% RSLogix 500 project I2P Hands-On 4 - Myah.RSS, saved by version 10.00.00.00 %
PROJECT "UNTITLED"    % processor: Bul.1763 MicroLogix 1100 Series B %

PROGRAM FILES
  LAD 2   15 rungs

DATA FILES
  O0 OUTPUT  4 elements
  I1 INPUT  6 elements
  S2 STATUS  66 elements
  B3 BINARY  1 elements
  T4 TIMER  1 elements
  C5 COUNTER  1 elements
  R6 CONTROL  1 elements
  N7 INTEGER  1 elements
  F8 FLOAT  1 elements

LADDER 2
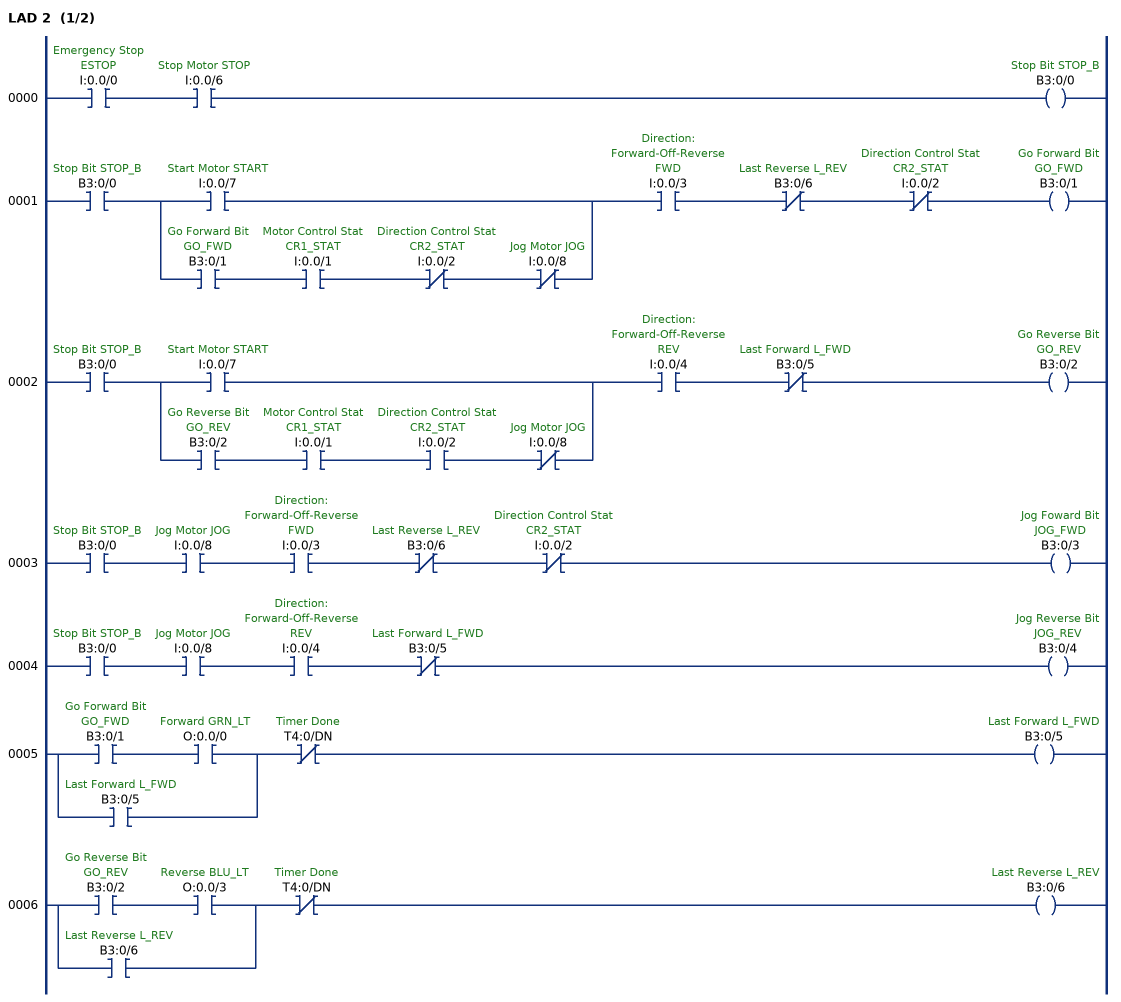
% Rung: 0 %
SOR XIC I:0.0/0 XIC I:0.0/6 OTE B3:0/0 EOR
%   I:0.0/0  ESTOP  "Emergency Stop" %
%   I:0.0/6  STOP  "Stop Motor" %
%   B3:0/0  STOP_B  "Stop Bit" %
% Rung: 1 %
SOR XIC B3:0/0 BST XIC I:0.0/7 NXB XIC B3:0/1 XIC I:0.0/1 XIO I:0.0/2 XIO I:0.0/8 BND XIC I:0.0/3 XIO B3:0/6 XIO I:0.0/2 OTE B3:0/1 EOR
%   B3:0/0  STOP_B  "Stop Bit" %
%   I:0.0/7  START  "Start Motor" %
%   B3:0/1  GO_FWD  "Go Forward Bit" %
%   I:0.0/1  CR1_STAT  "Motor Control Stat" %
%   I:0.0/2  CR2_STAT  "Direction Control Stat" %
%   I:0.0/8  JOG  "Jog Motor" %
%   I:0.0/3  FWD  "Direction: Forward-Off-Reverse" %
%   B3:0/6  L_REV  "Last Reverse" %
% Rung: 2 %
SOR XIC B3:0/0 BST XIC I:0.0/7 NXB XIC B3:0/2 XIC I:0.0/1 XIC I:0.0/2 XIO I:0.0/8 BND XIC I:0.0/4 XIO B3:0/5 OTE B3:0/2 EOR
%   B3:0/0  STOP_B  "Stop Bit" %
%   I:0.0/7  START  "Start Motor" %
%   B3:0/2  GO_REV  "Go Reverse Bit" %
%   I:0.0/1  CR1_STAT  "Motor Control Stat" %
%   I:0.0/2  CR2_STAT  "Direction Control Stat" %
%   I:0.0/8  JOG  "Jog Motor" %
%   I:0.0/4  REV  "Direction: Forward-Off-Reverse" %
%   B3:0/5  L_FWD  "Last Forward" %
% Rung: 3 %
SOR XIC B3:0/0 XIC I:0.0/8 XIC I:0.0/3 XIO B3:0/6 XIO I:0.0/2 OTE B3:0/3 EOR
%   B3:0/0  STOP_B  "Stop Bit" %
%   I:0.0/8  JOG  "Jog Motor" %
%   I:0.0/3  FWD  "Direction: Forward-Off-Reverse" %
%   B3:0/6  L_REV  "Last Reverse" %
%   I:0.0/2  CR2_STAT  "Direction Control Stat" %
%   B3:0/3  JOG_FWD  "Jog Foward Bit" %
% Rung: 4 %
SOR XIC B3:0/0 XIC I:0.0/8 XIC I:0.0/4 XIO B3:0/5 OTE B3:0/4 EOR
%   B3:0/0  STOP_B  "Stop Bit" %
%   I:0.0/8  JOG  "Jog Motor" %
%   I:0.0/4  REV  "Direction: Forward-Off-Reverse" %
%   B3:0/5  L_FWD  "Last Forward" %
%   B3:0/4  JOG_REV  "Jog Reverse Bit" %
% Rung: 5 %
SOR BST XIC B3:0/1 XIC O:0.0/0 NXB XIC B3:0/5 BND XIO T4:0/DN OTE B3:0/5 EOR
%   B3:0/1  GO_FWD  "Go Forward Bit" %
%   O:0.0/0  GRN_LT  "Forward" %
%   B3:0/5  L_FWD  "Last Forward" %
%   T4:0/DN  "Timer Done" %
% Rung: 6 %
SOR BST XIC B3:0/2 XIC O:0.0/3 NXB XIC B3:0/6 BND XIO T4:0/DN OTE B3:0/6 EOR
%   B3:0/2  GO_REV  "Go Reverse Bit" %
%   O:0.0/3  BLU_LT  "Reverse" %
%   B3:0/6  L_REV  "Last Reverse" %
%   T4:0/DN  "Timer Done" %

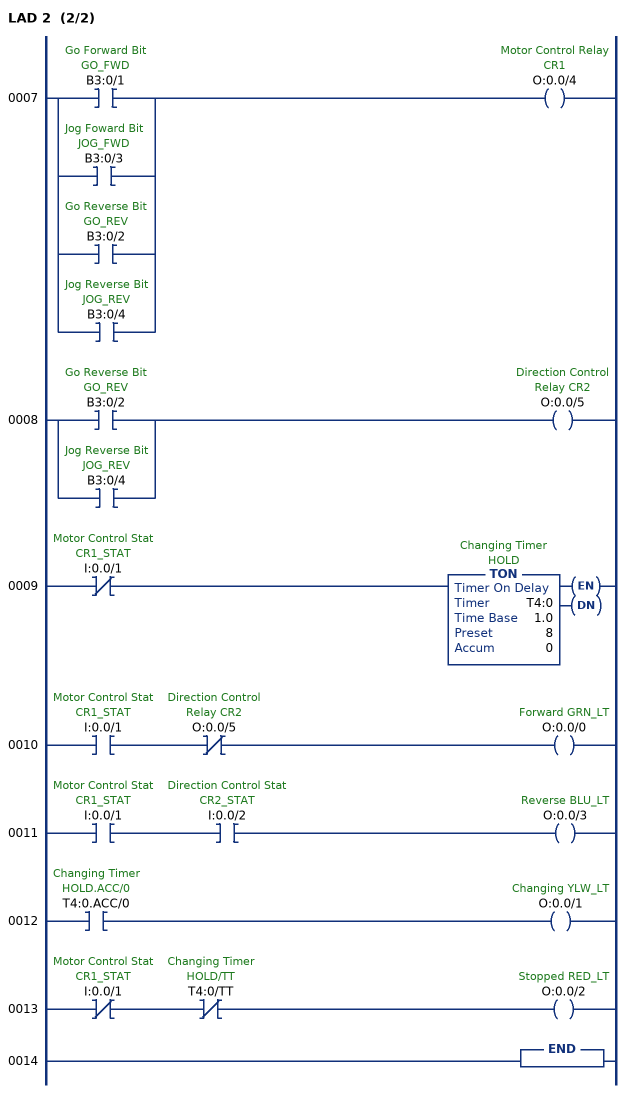
% Rung: 7 %
SOR BST XIC B3:0/1 NXB BST XIC B3:0/3 NXB BST XIC B3:0/2 NXB XIC B3:0/4 BND BND BND OTE O:0.0/4 EOR
%   B3:0/1  GO_FWD  "Go Forward Bit" %
%   B3:0/3  JOG_FWD  "Jog Foward Bit" %
%   B3:0/2  GO_REV  "Go Reverse Bit" %
%   B3:0/4  JOG_REV  "Jog Reverse Bit" %
%   O:0.0/4  CR1  "Motor Control Relay" %
% Rung: 8 %
SOR BST XIC B3:0/2 NXB XIC B3:0/4 BND OTE O:0.0/5 EOR
%   B3:0/2  GO_REV  "Go Reverse Bit" %
%   B3:0/4  JOG_REV  "Jog Reverse Bit" %
%   O:0.0/5  CR2  "Direction Control Relay" %
% Rung: 9 %
SOR XIO I:0.0/1 TON T4:0 1.0 8 0 EOR
%   I:0.0/1  CR1_STAT  "Motor Control Stat" %
%   T4:0  HOLD  "Changing Timer" %
% Rung: 10 %
SOR XIC I:0.0/1 XIO O:0.0/5 OTE O:0.0/0 EOR
%   I:0.0/1  CR1_STAT  "Motor Control Stat" %
%   O:0.0/5  CR2  "Direction Control Relay" %
%   O:0.0/0  GRN_LT  "Forward" %
% Rung: 11 %
SOR XIC I:0.0/1 XIC I:0.0/2 OTE O:0.0/3 EOR
%   I:0.0/1  CR1_STAT  "Motor Control Stat" %
%   I:0.0/2  CR2_STAT  "Direction Control Stat" %
%   O:0.0/3  BLU_LT  "Reverse" %
% Rung: 12 %
SOR XIC T4:0.ACC/0 OTE O:0.0/1 EOR
%   T4:0  HOLD  "Changing Timer" %
%   O:0.0/1  YLW_LT  "Changing" %
% Rung: 13 %
SOR XIO I:0.0/1 XIO T4:0/TT OTE O:0.0/2 EOR
%   I:0.0/1  CR1_STAT  "Motor Control Stat" %
%   T4:0  HOLD  "Changing Timer" %
%   O:0.0/2  RED_LT  "Stopped" %
% Rung: 14 %
SOR END EOR

DATA TABLE (non-zero values as saved)
DATA T4
% .PRE .ACC %
% T4:0 % 8 0
